Staubli VAL3: GetTrajFlag.pgx

public program GetTrajFlag(bool& x_bRes (dimensions=1), string x_sFileName (dimensions=1), num x_nTrajIndex (dimensions=1), num& x_nStart (dimensions=1), num& x_nEnd (dimensions=1))
  local string l_sBuff
  local num l_nIndex
  local num l_nStartIndex
  local num l_nEndIndex
begin
  //参数初始化
  x_bRes=false
  x_nStart=0
  x_nEnd=0
  l_sBuff=""
  l_nIndex=0
  l_nEndIndex=0
  l_nStartIndex=0

  //传入参数合法性判断
  if x_sFileName=="" or x_nTrajIndex<1
    return
  endIf

  //打开文件
  nFileID=$fileOpen(x_sFileName,"r")
  if nFileID<0 or nFileID>9
    return
  endIf


  //查询关键字
  while !x_bRes and $fileGet(nFileID,l_sBuff,1)==1
    l_nIndex=l_nIndex+1

    if find(l_sBuff,"=BEGIN")>=0
      l_nStartIndex=l_nStartIndex+1
      x_nStart=l_nIndex
    endIf

    if find(l_sBuff,"=END")>=0
      l_nEndIndex=l_nEndIndex+1
      x_nEnd=l_nIndex
    endIf

    if l_nStartIndex==x_nTrajIndex and l_nEndIndex==x_nTrajIndex

      x_bRes=true
    endIf

  endWhile

  call CloseAllFile()

  //把所有文件给关闭掉

end
